// TIA Portal V19 export
DATA_BLOCK "IF_Device"   // DB27
{ S7_Optimized_Access := 'TRUE' }
// stored: AutoNumber false, MemoryReserve 0
   VAR RETAIN
      TTX_09_30 : Struct   // IFM TA2502
         ProcessData : Struct
            Temperature : Real := 0.0;   // act. temperature [C]
         END_STRUCT;
         OP : "OP_Int";   // operating acyclic communication
         Commands : Struct   // commands interface
            Commando_1 : Bool;   // (1) Upload Start
            Commando_2 : Bool;   // (2) Upload End
            Commando_3 : Bool;   // (3) Download Start
            Commando_4 : Bool;   // (4) Download End
            Commando_5 : Bool;   // (5) Store
            Commando_6 : Bool;   // (6) Break
            Commando_7 : Bool;   // (130) Restore Factory Settings
            Commando_8 : Bool;   // (240) Test Event 8DFE appears
            Commando_9 : Bool;   // (241) Test Event 8DFE disappears
            Commando_10 : Bool;   // (242) Test Event 8DFF appears
            Commando_11 : Bool;   // (243) Test Event 8DFF disappears
            Commando_12 : Bool;   // not used
            Commando_13 : Bool;   // not used
            Commando_14 : Bool;   // not used
            Commando_15 : Bool;   // not used
            Commando_16 : Bool;   // not used
            Commando_17 : Bool;   // not used
            Commando_18 : Bool;   // not used
            Commando_19 : Bool;   // not used
            Commando_20 : Bool;   // not used
            Commando_21 : Bool;   // not used
            Commando_22 : Bool;   // not used
            Commando_23 : Bool;   // not used
            Commando_24 : Bool;   // not used
         END_STRUCT;
         "IF" : "IF_TA2502";
         PQI : "PQI_IF";   // PQI diagnostic information
      END_STRUCT;
      TTX_09_31 : Struct   // IFM TA2502
         ProcessData : Struct
            Temperature : Real := 0.0;   // act. temperature [C]
         END_STRUCT;
         OP : "OP_Int";   // operating acyclic communication
         Commands : Struct   // commands interface
            Commando_1 : Bool;   // (1) Upload Start
            Commando_2 : Bool;   // (2) Upload End
            Commando_3 : Bool;   // (3) Download Start
            Commando_4 : Bool;   // (4) Download End
            Commando_5 : Bool;   // (5) Store
            Commando_6 : Bool;   // (6) Break
            Commando_7 : Bool;   // (130) Restore Factory Settings
            Commando_8 : Bool;   // (240) Test Event 8DFE appears
            Commando_9 : Bool;   // (241) Test Event 8DFE disappears
            Commando_10 : Bool;   // (242) Test Event 8DFF appears
            Commando_11 : Bool;   // (243) Test Event 8DFF disappears
            Commando_12 : Bool;   // not used
            Commando_13 : Bool;   // not used
            Commando_14 : Bool;   // not used
            Commando_15 : Bool;   // not used
            Commando_16 : Bool;   // not used
            Commando_17 : Bool;   // not used
            Commando_18 : Bool;   // not used
            Commando_19 : Bool;   // not used
            Commando_20 : Bool;   // not used
            Commando_21 : Bool;   // not used
            Commando_22 : Bool;   // not used
            Commando_23 : Bool;   // not used
            Commando_24 : Bool;   // not used
         END_STRUCT;
         "IF" : "IF_TA2502";
         PQI : "PQI_IF";   // PQI diagnostic information
      END_STRUCT;
      CTX_09_30 : Struct   // IFM LDL101
         ProcessData : Struct
            Conductivity : Real := 0.0;   // act. conductivity [S]
            Temperature1 : Real := 0.0;   // act. temperature [C]
         END_STRUCT;
         OP : "OP_Int";   // operating acyclic communication
         Commands : Struct   // commands interface
            Commando_1 : Bool;   // (1) Upload Start
            Commando_2 : Bool;   // (2) Upload End
            Commando_3 : Bool;   // (3) Download Start
            Commando_4 : Bool;   // (4) Download End
            Commando_5 : Bool;   // (5) Store
            Commando_6 : Bool;   // (6) Break
            Commando_7 : Bool;   // (130) Restore Factory Settings
            Commando_8 : Bool;   // (240) Test Event 8DFE appears
            Commando_9 : Bool;   // (241) Test Event 8DFE disappears
            Commando_10 : Bool;   // (242) Test Event 8DFF appears
            Commando_11 : Bool;   // (243) Test Event 8DFF disappears
            Commando_12 : Bool;   // not used
            Commando_13 : Bool;   // not used
            Commando_14 : Bool;   // not used
            Commando_15 : Bool;   // not used
            Commando_16 : Bool;   // not used
            Commando_17 : Bool;   // not used
            Commando_18 : Bool;   // not used
            Commando_19 : Bool;   // not used
            Commando_20 : Bool;   // not used
            Commando_21 : Bool;   // not used
            Commando_22 : Bool;   // not used
            Commando_23 : Bool;   // not used
            Commando_24 : Bool;   // not used
         END_STRUCT;
         "IF" : "IF_LDL101";
         PQI : "PQI_IF";   // PQI diagnostic information
      END_STRUCT;
      V_09_30 : Struct   // Burkett CH Type 8691
         OP : "OP_Int";
         Commands : Struct   // commands interface
            Commando_1 : Bool;   // (128) Device Reset
            Commando_2 : Bool;   // (130) Restore Factory Settings
            Commando_3 : Bool;   // (160) Start Auto Teach function
            Commando_4 : Bool;   // (161) Start Manual Teach function
            Commando_5 : Bool;   // not used
            Commando_6 : Bool;   // not used
            Commando_7 : Bool;   // not used
            Commando_8 : Bool;   // not used
            Commando_9 : Bool;   // not used
            Commando_10 : Bool;   // not used
            Commando_11 : Bool;   // not used
            Commando_12 : Bool;   // not used
            Commando_13 : Bool;   // not used
            Commando_14 : Bool;   // not used
            Commando_15 : Bool;   // not used
            Commando_16 : Bool;   // not used
            Commando_17 : Bool;   // not used
            Commando_18 : Bool;   // not used
            Commando_19 : Bool;   // not used
            Commando_20 : Bool;   // not used
            Commando_21 : Bool;   // not used
            Commando_22 : Bool;   // not used
            Commando_23 : Bool;   // not used
            Commando_24 : Bool;   // not used
         END_STRUCT;
         IO : "IO Burkett Type 8691";
         "IF" : "IF Burkett Type 8691 IO";
      END_STRUCT;
      V_09_31 : Struct   // Burkett CH Type 8691
         OP : "OP_Int";
         Commands : Struct   // commands interface
            Commando_1 : Bool;   // (128) Device Reset
            Commando_2 : Bool;   // (130) Restore Factory Settings
            Commando_3 : Bool;   // (160) Start Auto Teach function
            Commando_4 : Bool;   // (161) Start Manual Teach function
            Commando_5 : Bool;   // not used
            Commando_6 : Bool;   // not used
            Commando_7 : Bool;   // not used
            Commando_8 : Bool;   // not used
            Commando_9 : Bool;   // not used
            Commando_10 : Bool;   // not used
            Commando_11 : Bool;   // not used
            Commando_12 : Bool;   // not used
            Commando_13 : Bool;   // not used
            Commando_14 : Bool;   // not used
            Commando_15 : Bool;   // not used
            Commando_16 : Bool;   // not used
            Commando_17 : Bool;   // not used
            Commando_18 : Bool;   // not used
            Commando_19 : Bool;   // not used
            Commando_20 : Bool;   // not used
            Commando_21 : Bool;   // not used
            Commando_22 : Bool;   // not used
            Commando_23 : Bool;   // not used
            Commando_24 : Bool;   // not used
         END_STRUCT;
         IO : "IO Burkett Type 8691";
         "IF" : "IF Burkett Type 8691 IO";
      END_STRUCT;
   END_VAR
BEGIN
   TTX_09_30.OP.I_DataStorage := TRUE;
   TTX_09_30.OP.I_BlockParam := TRUE;
   TTX_09_31.OP.I_DataStorage := TRUE;
   TTX_09_31.OP.I_BlockParam := TRUE;
   CTX_09_30.OP.I_DataStorage := TRUE;
   CTX_09_30.OP.I_BlockParam := TRUE;
   V_09_30.OP.I_DataStorage := TRUE;
   V_09_30.OP.I_BlockParam := TRUE;
   V_09_30.IO.V._IO.OUT.ValvePosition := 0.0;
   V_09_30."IF".StandardStructure.DeviceParameters.Parameter_08.Value.UpperEndPosition := 0.0;
   V_09_30."IF".StandardStructure.DeviceParameters.Parameter_09.Value.LowerEndPosition := 0.0;
   V_09_30."IF".StandardStructure.DeviceParameters.Parameter_12.Value.Stroke := 0.0;
   V_09_30."IF".StandardStructure.DeviceParameters.Parameter_20.Value.TravelAccumlator := 0.0;
   V_09_30."IF".StandardStructure.DeviceParameters.Parameter_21.Value.TravelAccResettable := 0.0;
   V_09_30."IF".StandardStructure.DeviceParameters.Parameter_22.Value.TravelAccLimit := 0.0;
   V_09_30."IF".StandardStructure.DeviceParameters.Parameter_29.Value.OpeningTimeLimit := 2000;
   V_09_30."IF".StandardStructure.DeviceParameters.Parameter_30.Value.ClosingTimeLimit := 2000;
   V_09_30."IF".StandardStructure.DeviceParameters.Parameter_31.Value.TimeTolerance := BYTE#16#0A;
   V_09_30."IF".StandardStructure.DeviceParameters.Parameter_39.Value.SwitchingTimeout := 3000;
   V_09_31.OP.I_DataStorage := TRUE;
   V_09_31.OP.I_BlockParam := TRUE;
   V_09_31.IO.V._IO.OUT.ValvePosition := 0.0;
   V_09_31."IF".StandardStructure.DeviceParameters.Parameter_08.Value.UpperEndPosition := 0.0;
   V_09_31."IF".StandardStructure.DeviceParameters.Parameter_09.Value.LowerEndPosition := 0.0;
   V_09_31."IF".StandardStructure.DeviceParameters.Parameter_12.Value.Stroke := 0.0;
   V_09_31."IF".StandardStructure.DeviceParameters.Parameter_20.Value.TravelAccumlator := 0.0;
   V_09_31."IF".StandardStructure.DeviceParameters.Parameter_21.Value.TravelAccResettable := 0.0;
   V_09_31."IF".StandardStructure.DeviceParameters.Parameter_22.Value.TravelAccLimit := 0.0;
   V_09_31."IF".StandardStructure.DeviceParameters.Parameter_29.Value.OpeningTimeLimit := 2000;
   V_09_31."IF".StandardStructure.DeviceParameters.Parameter_30.Value.ClosingTimeLimit := 2000;
   V_09_31."IF".StandardStructure.DeviceParameters.Parameter_31.Value.TimeTolerance := BYTE#16#0A;
   V_09_31."IF".StandardStructure.DeviceParameters.Parameter_39.Value.SwitchingTimeout := 3000;
END_DATA_BLOCK
